# EPICS StreamDevice protocol: CalSysSup/BO-CalSys.proto
ReplyTimeout=1000;
ReadTimeout=1000;

getData {
    InTerminator=CR LF;
    separator=', ';
    ExtraInput=Ignore;
    out "ADC0:DATA?";
    in  "[%f]";
}
